// TwinCAT 3 PLC project MotionRewrite1
// ProgramVersion: 3.1.4023.0
// libraries:
//   Tc2_MC2, * (Beckhoff Automation GmbH)
//   Tc2_Standard, * (Beckhoff Automation GmbH)
//   Tc2_System, * (Beckhoff Automation GmbH)
//   Tc3_Module, * (Beckhoff Automation GmbH)
// project tree:
//   DUTs/Abstract/Linear/ I_LinearContinuousDrive.TcIO, I_LinearDrive.TcIO (not stored), I_LinearEncodedDrive.TcIO
//   DUTs/Drives - Generic/ AirPiston.TcPOU (not stored), ClearLinkMC.TcPOU, ServoNC.TcPOU
//   DUTs/Drives - Linear/ LinearContinuousDrive_2Sensor.TcPOU, LinearEncodedDrive_2Sensor.TcPOU (not stored), LinearEncodedDrive_3Sensor.TcPOU, LinearContinuousDrive_3Sensor.TcPOU (not stored)
//   DUTs/Insertion Package/ Homing.TcDUT (not stored), Insertion.TcPOU (not stored), Insertion2D.TcPOU (not stored), SuctionPad.TcDUT (not stored)
//   DUTs/Abstract/ FBA_LinearDrive.TcPOU, I_ContinuousDrive.TcIO (not stored), I_Drive.TcIO, I_EncodedDrive.TcIO (not stored), I_PositionalDrive.TcIO
//   / PlcTask.TcTTO (not stored)
//   POUs/ MAIN.TcPOU (not stored), WithinTolerance.TcPOU (not stored)
// real-time tasks:
//   TASK PlcTask: cycle T#10ms, priority 33, ADS port 350
//   TASK PlcTask1: cycle T#10ms, priority 20, ADS port 351

// ---- DUTs/Abstract/Linear/I_LinearContinuousDrive.TcIO
INTERFACE I_LinearContinuousDrive EXTENDS I_LinearDrive, I_ContinuousDrive

END_INTERFACE

// ---- DUTs/Abstract/Linear/I_LinearEncodedDrive.TcIO
INTERFACE I_LinearEncodedDrive EXTENDS I_LinearContinuousDrive, I_EncodedDrive

END_INTERFACE

// ---- DUTs/Abstract/I_Drive.TcIO
INTERFACE I_Drive

{attribute 'monitoring':='call'}
PROPERTY Active : BOOL
GET
END_GET
END_PROPERTY

{attribute 'monitoring':='call'}
PROPERTY Error : BOOL
GET
END_GET
END_PROPERTY

METHOD reset : BOOL
VAR_INPUT
END_VAR
END_METHOD

METHOD ABSTRACT stop : BOOL
VAR_INPUT
END_VAR
END_METHOD

END_INTERFACE

// ---- DUTs/Abstract/I_PositionalDrive.TcIO
INTERFACE I_PositionalDrive EXTENDS I_Drive

PROPERTY CurrentPosition : LREAL
GET
END_GET
END_PROPERTY

METHOD ABSTRACT moveAbsolute : BOOL
VAR_INPUT
	newTarget : LREAL; 
END_VAR
END_METHOD

METHOD ABSTRACT moveRelative : BOOL
VAR_INPUT
	distance : LREAL;
END_VAR
END_METHOD

METHOD setPosition : BOOL
VAR_INPUT
	newPosition : LREAL;
END_VAR
END_METHOD

PROPERTY TargetPosition : LREAL
GET
END_GET
END_PROPERTY

END_INTERFACE

// ---- DUTs/Drives - Generic/ClearLinkMC.TcPOU
FUNCTION_BLOCK ClearLinkMC IMPLEMENTS I_EncodedDrive
VAR_INPUT
	bEnable : BOOL;
END_VAR
VAR_OUTPUT
	pulse AT %Q* : INT;
	brakeRelease AT %Q* : BOOL := TRUE;
	enable : BOOL;
	A : BOOL;
	B : BOOL;
	clear : BOOL;
END_VAR
VAR	
	hlfb AT %I* : REAL := -9999; //high level feedback, if -9999 then servo is idle
	
	outputRegister AT %Q* : INT;
	pulseRequest : INT;
	
	homingDelay : TON;
	resetPulse : TP;
	
	mode : (HOLD, TARGET, CONTINUOUS, RESET_ERR);
	calculation : (IDLE, DOWN, UP, CALCULATE, DONE);
	maxPosition : LREAL;
	
	position, targetPos : LREAL;
	
	pulsePosition : INT;
	pulseCounter : INT;
	rotationsPerPulse : INT; //revolutions per pulse
	displacementPerPulse : LREAL; //displacement per pulse
END_VAR
VAR_STAT CONSTANT
	resetWidth : TIME := T#500MS;
	delayWidth : TIME := T#500MS;
END_VAR
VAR //constructor
	homingDirectionOut : BOOL; 			//homing direction - see <A>
	minPosition : LREAL;
	displacementPerRotation : LREAL; 	//displacement per revolution	
	unitsPerPulse : INT := 800; 		//800 Teknic units per rotation - default setting is 800 units (1 rotation) per pulse
END_VAR

//M-connector output register
outputRegister.0 := enable AND bEnable; 	//enable
outputRegister.1 := A; 						//direction bit - T = outwards, F = inwards
outputRegister.2 := B; 						//homing bit - after startup, set to TRUE to begin homing, then set to FALSE to finish homing
outputRegister.3 := clear; 					//reset bit

rotationsPerPulse := unitsPerPulse/800; //Teknic constant - 800 units per rotation
displacementPerPulse := displacementPerRotation * rotationsPerPulse;

resetPulse(IN:= , PT:= resetWidth, Q=> clear, ET=> ); //reset pulse

IF NOT enable THEN
	stop();
END_IF

override();

CASE mode OF		
	HOLD: //hold current position, no motion
		pulse := 0;
		pulseRequest := 0;
	
	TARGET:	//target a given position
		
		IF WithinTolerance(position, targetPos, displacementPerPulse) THEN
			pulseRequest := 0;
			pulse := 0;
			mode := HOLD;
			
		ELSIF NOT Active THEN
			A :=  position < targetPos;
			(*
			2 options to traverse to a target position:
				a)  send all pulses at once - continuous motion but may exceed limits, check for bounds before setting
				b)  1 pulse at a time - choppy but safer
			*)
			targetPos := MAX(targetPos, minPosition); //if below minPosition, set to minPosition
			targetPos := MIN(targetPos, maxPosition); //if above maxPosition, set to maxPosition
			
			pulseRequest := TO_INT(ABS(position - targetPos)/displacementPerPulse);
			//pulseRequest := 1;
		END_IF
		
	CONTINUOUS: //single pulses in the direction specified by moveContinuous()
		pulseRequest := 1;
		
	RESET_ERR: //reset pulse, servo may need to be rehomed aftewards
		pulse := 0;
		pulseRequest := 0;
		resetPulse.IN := TRUE;
		
		IF resetPulse.Q THEN
			resetPulse.IN := FALSE;
			mode := HOLD;
		END_IF
		
END_CASE

sequence();

PROPERTY Active : BOOL
GET
Active := hlfb <> -9999;
END_GET
END_PROPERTY

PROPERTY CurrentPosition : LREAL
GET
CurrentPosition := position;

//CurrentPosition := pulsePosition * displacementPerPulse;
END_GET
SET
position := CurrentPosition;
END_SET
END_PROPERTY

PROPERTY Error : BOOL
GET
END_GET
END_PROPERTY

{attribute 'TcRpcEnable'}
METHOD moveAbsolute : BOOL
VAR_INPUT
	newTarget : LREAL;
END_VAR
IF target >= maxPosition AND target <= minPosition THEN
	A :=  position < targetPos;
	targetPos := newTarget;
	mode := TARGET;
	
	moveAbsolute := TRUE;
END_IF
END_METHOD

{attribute 'TcRpcEnable'}
METHOD moveContinuous : BOOL
VAR_INPUT
	newDirection : MC_Direction;
END_VAR
IF newDirection = MC_Negative_Direction THEN
	A := FALSE;
ELSIF newDirection = MC_Positive_Direction THEN
	A := TRUE;
END_IF

mode := CONTINUOUS;
END_METHOD

{attribute 'TcRpcEnable'}
METHOD moveRelative : BOOL
VAR_INPUT
	distance : LREAL;
END_VAR
targetPos := targetPos + distance;

mode := TARGET;
END_METHOD

METHOD PRIVATE override : BOOL
VAR_INPUT
END_VAR
IF error THEN
	stop();
	reset();
END_IF

(*
IF AtHome AND NOT Active THEN
	IF homingDirectionOut THEN //homing is outwards
		position := maxPosition;
		pulsePosition := pulseCounter;
	ELSE
		position := minPosition;
		pulsePosition := 0;
	END_IF
	

ELSIF AtInnerLimit AND NOT Active THEN
	IF homingDirectionOut THEN //homing is outwards
		position := minPosition;
		pulsePosition := 0;
	ELSE
		position := maxPosition;
		pulsePosition := pulseCounter;
	END_IF
END_IF

CASE mode OF		
	HOLD:
		//
	
	TARGET:
		IF
			(AtHome AND TargetPosition > CurrentPosition) OR
			(AtInnerLimit AND TargetPosition > CurrentPosition) OR
			(AtOuterLimit AND TargetPosition < CurrentPosition)
		THEN
			mode := HOLD;
		END_IF
		
	CONTINUOUS:
		IF
			(AtHome AND A) OR
			(AtInnerLimit AND A) OR
			(AtOuterLimit AND NOT A)
		THEN
			mode := HOLD;
		END_IF
		
	RESET_ERR:
		//
		
END_CASE
*)
END_METHOD

METHOD reset : BOOL
VAR_INPUT
END_VAR
mode := RESET_ERR;
END_METHOD

METHOD PRIVATE sequence : BOOL
VAR_INPUT
END_VAR
IF Active THEN //servo is active
	IF A THEN //positive direction
		position := position + (displacementPerPulse * pulse);
		pulsePosition := pulsePosition + pulse;
		
		pulseCounter := pulseCounter + pulse;
	ELSE //negative direction
		position := position - (displacementPerPulse * pulse);
		pulsePosition := pulsePosition - pulse;
		
		pulseCounter := pulseCounter - pulse;
	END_IF
	pulse := 0; //pulses already received, can be set to 0 so position change is not compounded

ELSIF pulse = 0 THEN //servo is not active
	pulse := pulseRequest;
END_IF

pulseRequest := 0; //remove this if not working as intended
END_METHOD

METHOD setPosition : BOOL
VAR_INPUT
	newPosition : LREAL;
END_VAR
position := newPosition;

setPosition := position = newPosition;
END_METHOD

METHOD stop : BOOL
VAR_INPUT
END_VAR
mode := HOLD;
END_METHOD

PROPERTY TargetPosition : LREAL
GET
END_GET
SET
targetPos := TargetPosition;
END_SET
END_PROPERTY

END_FUNCTION_BLOCK

// ---- DUTs/Drives - Generic/ServoNC.TcPOU
FUNCTION_BLOCK ServoNC IMPLEMENTS I_EncodedDrive
VAR_INPUT
	bEnable : BOOL;
END_VAR
VAR_OUTPUT	
	ready : BOOL;
	position : LREAL;
	velocity : LREAL;
END_VAR
VAR
	axis : AXIS_REF;
	
	mcReadPosition : MC_ReadActualPosition; //continuous enable FBs
	mcReadVelocity : MC_ReadActualVelocity;
	mcReadError : MC_ReadAxisError;
	mcPower : MC_Power;
	
	mcReset : MC_Reset; //rising edge FBs
	mcMoveAbsolute : MC_MoveAbsolute;
	mcMoveRelative : MC_MoveRelative;
	mcMoveVelocity : MC_MoveVelocity;
	
	mcSetPosition : MC_SetPosition;
	mcStop : MC_Stop;
END_VAR
VAR_STAT CONSTANT
	targetingVelocity : INT := 500;
	continuousVelocity : INT := 100;
END_VAR

override();

blocks();

mcReset.Execute := FALSE;
mcMoveAbsolute.Execute := FALSE;
mcMoveRelative.Execute := FALSE;
mcMoveVelocity.Execute := FALSE;
mcSetPosition.Execute := FALSE;
mcStop.Execute := FALSE;

blocks();

ready := bEnable AND NOT Active;

PROPERTY Active : BOOL
GET
Active := 
	mcMoveAbsolute.Busy OR 
	mcMoveRelative.Busy OR 
	mcMoveVelocity.Busy OR 
	mcSetPosition.Busy OR 
	mcReset.Busy OR 
	mcStop.Busy;
END_GET
END_PROPERTY

METHOD PRIVATE blocks : BOOL
mcReadPosition(
	Axis:= axis, 
	Enable:= TRUE, 
	Valid=> , 
	Busy=> , 
	Error=> , 
	ErrorID=> , 
	Position=> position);
	
mcReadVelocity(
	Axis:= axis, 
	Enable:= TRUE, 
	Valid=> , 
	Busy=> , 
	Error=> , 
	ErrorID=> , 
	ActualVelocity=> velocity);
	
mcReadError(
	Axis:= axis, 
	Enable:= TRUE, 
	Valid=> , 
	Busy=> , 
	Error=> , 
	ErrorID=> , 
	AxisErrorID=> );

mcReset(
	Axis:= axis, 
	Execute:= , 
	Done=> , 
	Busy=> , 
	Error=> , 
	ErrorID=> );

mcPower(
	Axis:= axis, 
	Enable:= bEnable, 
	Enable_Positive:= TRUE, 
	Enable_Negative:= TRUE, 
	Override:= 100, 
	BufferMode:= , 
	Options:= , 
	Status=> , 
	Busy=> , 
	Active=> , 
	Error=> , 
	ErrorID=> );

mcMoveAbsolute(
	Axis:= axis, 
	Execute:= , 
	Position:= , 
	Velocity:= targetingVelocity, 
	Acceleration:= , 
	Deceleration:= , 
	Jerk:= , 
	BufferMode:= , 
	Options:= , 
	Done=> , 
	Busy=> , 
	Active=> , 
	CommandAborted=> , 
	Error=> , 
	ErrorID=> );
	
mcMoveRelative(
	Axis:= axis, 
	Execute:= , 
	Distance:= ,
	Velocity:= targetingVelocity, 
	Acceleration:= , 
	Deceleration:= , 
	Jerk:= , 
	BufferMode:= , 
	Options:= , 
	Done=> , 
	Busy=> , 
	Active=> , 
	CommandAborted=> , 
	Error=> , 
	ErrorID=> );
	
mcMoveVelocity( //stopped with stop();
	Axis:= axis, 
	Execute:= , 
	Velocity:= continuousVelocity, 
	Acceleration:= , 
	Deceleration:= , 
	Jerk:= , 
	Direction:= , 
	BufferMode:= , 
	Options:= , 
	InVelocity=> , 
	Busy=> , 
	Active=> , 
	CommandAborted=> , 
	Error=> , 
	ErrorID=> );
	
mcSetPosition(
	Axis:= axis, 
	Execute:= , 
	Position:= , 
	Mode:= , 
	Options:= , 
	Done=> , 
	Busy=> , 
	Error=> , 
	ErrorID=> );
	
mcStop(
	Axis:= axis, 
	Execute:= , 
	Deceleration:= , 
	Jerk:= , 
	Options:= , 
	Done=> , 
	Busy=> , 
	Active=> , 
	CommandAborted=> , 
	Error=> , 
	ErrorID=> );
END_METHOD

PROPERTY CurrentPosition : LREAL
GET
CurrentPosition := position;
END_GET
SET
position := CurrentPosition;
END_SET
END_PROPERTY

PROPERTY Error : BOOL
GET
error := 
	mcMoveAbsolute.Error OR 
	mcMoveRelative.Error OR 
	mcMoveVelocity.Error OR 
	mcSetPosition.Error OR 
	mcReset.Error OR 
	mcStop.Error OR
	mcReadError.AxisErrorID > 0;
END_GET
END_PROPERTY

METHOD moveAbsolute : BOOL
VAR_INPUT
	newTarget : LREAL;
END_VAR
(*
VAR_OUTPUT
	fault : BOOL;
END_VAR
*)
IF NOT Active AND NOT error THEN
	mcMoveAbsolute.Position := newTarget;
	mcMoveAbsolute.Execute := TRUE;
END_IF

moveAbsolute := (*mcMoveAbsolute.Done AND mcMoveAbsolute.Active;*)
	position = newTarget;
END_METHOD

METHOD moveContinuous : BOOL
VAR_INPUT
	//direction : BOOL; //direction (F = inwards, T = outwards)
	newDirection : MC_Direction;
END_VAR
(*
IF mcMoveVelocity.Active THEN
	stop();
END_IF

IF NOT mcStop.Done THEN
	RETURN;
END_IF
*)
(*
IF direction THEN
	mcMoveVelocity.Direction := MC_Positive_Direction;
ELSE
	mcMoveVelocity.Direction := MC_Negative_Direction;
END_IF
*)
mcMoveVelocity.Direction := newDirection;

IF NOT mcMoveVelocity.Error THEN
	mcMoveVelocity.Execute := TRUE;
	moveContinuous := TRUE;
END_IF
END_METHOD

METHOD moveRelative : BOOL
VAR_INPUT
	distance : LREAL;
END_VAR
mcMoveRelative.Distance := distance;

moveRelative := mcMoveRelative.Done;
END_METHOD

METHOD PRIVATE override : BOOL
VAR_INPUT
END_VAR
IF error THEN
	stop();
	reset();
END_IF
END_METHOD

METHOD reset : BOOL
VAR_INPUT
END_VAR
mcReset.Execute := TRUE;

reset := mcReset.Done;
END_METHOD

METHOD setPosition : BOOL
VAR_INPUT
	newPosition : LREAL;
END_VAR
mcSetPosition.Position := newPosition;
mcSetPosition.Execute := TRUE;

setPosition := position = newPosition;
END_METHOD

METHOD stop : BOOL
VAR_INPUT
END_VAR
mcStop.Execute := TRUE;

mcMoveAbsolute.Execute := FALSE;
mcMoveRelative.Execute := FALSE;
mcMoveVelocity.Execute := FALSE;

stop := velocity = 0;
END_METHOD

PROPERTY TargetPosition : LREAL
GET
END_GET
SET
moveAbsolute(newTarget := TargetPosition);
END_SET
END_PROPERTY

END_FUNCTION_BLOCK

// ---- DUTs/Drives - Linear/LinearContinuousDrive_2Sensor.TcPOU
FUNCTION_BLOCK LinearContinuousDrive_2Sensor EXTENDS FBA_LinearDrive IMPLEMENTS I_LinearContinuousDrive
VAR_INPUT
	drive : I_ContinuousDrive;
END_VAR
VAR
	extendLimit AT %I* : BOOL;
END_VAR

override();

ready := bEnable AND NOT Active AND HomeSet;

PROPERTY Active : BOOL
GET
Active := drive.Active;
END_GET
END_PROPERTY

PROPERTY AtExtendLimit : BOOL
GET
AtExtendLimit := extendLimit <> sensorDefaultState;
END_GET
END_PROPERTY

PROPERTY Error : BOOL
GET
error := drive.Error;
END_GET
END_PROPERTY

METHOD homingSequence : BOOL
(*
homing sequence is different for linear motion devices with limit sensors
*)
CASE step OF
	Homing.IDLE:
		reset();
		IF bEnable THEN
			step := Homing.START;
		END_IF
		
	Homing.START:
		IF AtHome THEN
			step := Homing.STOP;
			
		ELSIF AtExtendLimit THEN
			step := Homing.RETRY;
			
		ELSE
			moveContinuous(newDirection:= MC_Positive_Direction);
		END_IF
		
	Homing.STOP:
		IF stop() THEN
			step := Homing.DONE;
		END_IF
		
	Homing.DONE:
		homingComplete := TRUE;
		step := Homing.IDLE;
		
END_CASE
END_METHOD

METHOD moveContinuous : BOOL
VAR_INPUT
	newDirection : MC_Direction;
END_VAR
drive.moveContinuous(newDirection:= newDirection);

direction := newDirection;
END_METHOD

METHOD PRIVATE override : BOOL
VAR_INPUT
END_VAR
(*
-at home and attempting to traverse outward
-at outer limit and attempting to traverse outward
-at inner limit and attempting to traverse inwards
*)
(*
inward = negative direction, negative velocity
outward = positive direction, positive velocity
*)

IF error THEN
	stop();
	reset();
	
ELSIF
	(AtExtendLimit AND direction = MC_Negative_Direction) OR
	(AtHome AND direction = MC_Positive_Direction)
THEN
	stop();
END_IF
END_METHOD

METHOD reset : BOOL
VAR_INPUT
END_VAR
reset := drive.reset();
END_METHOD

METHOD stop : BOOL
VAR_INPUT
END_VAR
stop := drive.stop();
END_METHOD

METHOD toHome : BOOL
VAR_INPUT
END_VAR
IF AtHome THEN
	toHome := TRUE;
ELSE
	moveContinuous(newDirection := MC_Negative_Direction);
END_IF
END_METHOD

END_FUNCTION_BLOCK

// ---- DUTs/Abstract/FBA_LinearDrive.TcPOU
FUNCTION_BLOCK ABSTRACT FBA_LinearDrive IMPLEMENTS I_LinearDrive
VAR_INPUT
	bEnable : BOOL;
	sensorDefaultState : BOOL;
END_VAR
VAR_OUTPUT	
	ready : BOOL;
END_VAR
VAR
	direction : MC_Direction;
	
	step : Homing;
	homingComplete : BOOL;
	
	home AT %I* : BOOL;
END_VAR

PROPERTY ABSTRACT Active : BOOL
GET
END_GET
END_PROPERTY

{attribute 'monitoring':='call'}
PROPERTY AtHome : BOOL
GET
AtHome := home <> sensorDefaultState;
END_GET
END_PROPERTY

PROPERTY ABSTRACT Error : BOOL
GET
END_GET
END_PROPERTY

{attribute 'monitoring':='call'}
PROPERTY HomeSet : BOOL
GET
HomeSet := homingComplete;
END_GET
END_PROPERTY

METHOD ABSTRACT homingSequence : BOOL
VAR_INPUT
END_VAR
END_METHOD

METHOD ABSTRACT reset : BOOL
VAR_INPUT
END_VAR
END_METHOD

METHOD ABSTRACT stop : BOOL
VAR_INPUT
END_VAR
END_METHOD

METHOD ABSTRACT toHome : BOOL
VAR_INPUT
END_VAR
END_METHOD

END_FUNCTION_BLOCK

// ---- DUTs/Drives - Linear/LinearEncodedDrive_3Sensor.TcPOU
FUNCTION_BLOCK LinearEncodedDrive_3Sensor EXTENDS FBA_LinearDrive IMPLEMENTS I_LinearEncodedDrive
VAR_INPUT
	drive : I_EncodedDrive;
	homeAt0 : BOOL;
	allowDualSideTraverse : BOOL; //allows motion between home to retractLimit
END_VAR
VAR_OUTPUT
	position : LREAL;
	velocity : LREAL;
END_VAR
VAR
	extendLimit AT %I* : BOOL;
	retractLimit AT %I* : BOOL;
	
	homePosition : LREAL;
	limitPosition : LREAL;
	
	calculation : (IDLE, EXTEND, RETRACT, CALCULATE, DONE);
END_VAR

override();

ready := bEnable AND NOT Active AND HomeSet;

PROPERTY Active : BOOL
GET
Active := drive.Active;
END_GET
END_PROPERTY

PROPERTY AtExtendLimit : BOOL
GET
AtExtendLimit := extendLimit <> sensorDefaultState;
END_GET
END_PROPERTY

PROPERTY AtRetractLimit : BOOL
GET
AtRetractLimit := retractLimit <> sensorDefaultState;
END_GET
END_PROPERTY

METHOD PRIVATE calculatePositions : BOOL
(*
THIS METHOD IS ONLY TO BE CALLED IF homeAt0 IS FALSE

not all drives have their home sensor at the 0 position
the purpose of this method is to calculate the home position, under the assumption that the extend limit sensor is 0

implementation:
	start from home
	reach the extend limit and set position to 0
	return to the home sensor and set the home position to the current position
*)
CASE calculation OF
	IDLE:
		calculation := EXTEND;
		
	EXTEND:		
		IF AtExtendLimit THEN
			
			IF homeAt0 THEN
				limitPosition := CurrentPosition;
				calculation := RETRACT;
			
			ELSIF setPosition(newPosition := 0) THEN
				limitPosition := 0;
				calculation := RETRACT;
			END_IF
		
		ELSE
			moveContinuous(newDirection := MC_Negative_Direction);
		END_IF
		
	RETRACT:
		IF AtHome THEN
			
			IF homeAt0 THEN
				homePosition := 0;
				calculation := DONE;
			
			ELSE
				homePosition := CurrentPosition;
				calculation := DONE;
			END_IF
		
		ELSE
			moveContinuous(newDirection := MC_Positive_Direction);
		END_IF
		
	DONE:
		calculation := 0;
		calculatePositions := TRUE;
		
END_CASE
END_METHOD

PROPERTY CurrentPosition : LREAL
GET
CurrentPosition := position;
END_GET
END_PROPERTY

PROPERTY Error : BOOL
GET
error := drive.Error;
END_GET
END_PROPERTY

METHOD homingSequence : BOOL
(*
homing sequence is different for linear motion devices with limit sensors
*)
CASE step OF
	Homing.IDLE:
		reset();
		IF bEnable THEN
			step := Homing.RETRY;
		END_IF
		
	Homing.START:
		IF AtHome THEN
			step := Homing.STOP;
			
		ELSIF AtRetractLimit THEN
			step := Homing.RETRY;
			
		ELSE
			moveContinuous(newDirection:= MC_Positive_Direction);
		END_IF
		
	Homing.RETRY:
		IF AtExtendLimit THEN
			step := Homing.START;
		ELSE
			moveContinuous(newDirection:= MC_Positive_Direction);
		END_IF
		
	Homing.STOP:
		IF stop() THEN
			step := Homing.SET;
		END_IF
		
	Homing.SET:
		IF calculatePositions() THEN
			step := Homing.DONE;
		END_IF
		
	Homing.DONE:
		homingComplete := TRUE;
		step := Homing.IDLE;
		
END_CASE
END_METHOD

METHOD moveAbsolute : BOOL
VAR_INPUT
	newTarget : LREAL;
END_VAR
(*
VAR_OUTPUT
	fault : BOOL;
END_VAR
*)
drive.moveAbsolute(newTarget:= newTarget);

moveAbsolute := drive.CurrentPosition = newTarget;
END_METHOD

METHOD moveContinuous : BOOL
VAR_INPUT
	//direction : BOOL; //direction (F = inwards, T = outwards)
	newDirection : MC_Direction;
END_VAR
drive.moveContinuous(newDirection:= newDirection);

direction := newDirection;
END_METHOD

METHOD moveRelative : BOOL
VAR_INPUT
	distance : LREAL;
END_VAR
drive.moveRelative(distance:= distance);
END_METHOD

METHOD PRIVATE override : BOOL
VAR_INPUT
END_VAR
(*
-at home and attempting to traverse outward
-at outer limit and attempting to traverse outward
-at inner limit and attempting to traverse inwards
*)
(*
inward = negative direction, negative velocity
outward = positive direction, positive velocity
*)

IF error THEN
	stop();
	reset();
	
ELSIF
	(NOT allowDualSideTraverse AND AtHome AND (TargetPosition > CurrentPosition OR direction = MC_Positive_Direction)) OR
	(AtExtendLimit AND (TargetPosition > CurrentPosition OR direction = MC_Negative_Direction)) OR
	(AtRetractLimit AND (TargetPosition < CurrentPosition OR direction = MC_Positive_Direction))
THEN
	stop();
END_IF
END_METHOD

METHOD reset : BOOL
VAR_INPUT
END_VAR
reset := drive.reset();
END_METHOD

METHOD setPosition : BOOL
VAR_INPUT
	newPosition : LREAL;
END_VAR
setPosition := drive.setPosition(newPosition:= newPosition);
END_METHOD

METHOD stop : BOOL
VAR_INPUT
END_VAR
drive.stop();
END_METHOD

PROPERTY TargetPosition : LREAL
GET
END_GET
END_PROPERTY

METHOD toHome : BOOL
VAR_INPUT
END_VAR
moveAbsolute(newTarget := homePosition);
END_METHOD

END_FUNCTION_BLOCK
